(* PLC project Unnamed, Unknown Unnamed 1 *)
(* stored: creationDateTime 2025-10-16T09:35:51, modificationDateTime 2025-10-21T14:08:54 *)

PROGRAM motor_ctrl
  VAR
    motor_error AT %IX0.0 : BOOL;
    motor_error_true AT %IX0.1 : BOOL;
    run_motor AT %QX0.0 : BOOL;
    motor_running AT %QX0.1 : BOOL;
    stop_motor AT %QX0.2 : BOOL;
    run_motor_true AT %QX0.3 : BOOL;
    motor_running_true AT %QX0.4 : BOOL;
    stop_motor_true AT %QX0.5 : BOOL;
    motor_rpm AT %IW0 : INT;
    motor_rpm_true AT %IW1 : INT;
    target_freq AT %QW0 : INT;
    target_freq_true AT %QW1 : INT := 120;
  END_VAR
  VAR  (* added by the conversion: wires and edge detectors of the diagram *)
    R_TRIG1 : R_TRIG;
    R_TRIG2 : R_TRIG;
  END_VAR

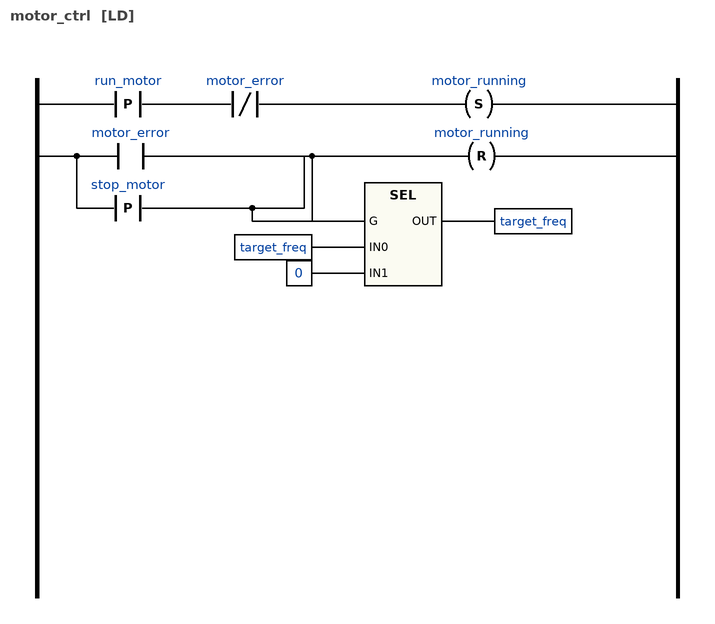
(* LD diagram, written out as Structured Text *)
R_TRIG1(CLK := run_motor);
IF R_TRIG1.Q AND NOT motor_error THEN motor_running := TRUE; END_IF;
R_TRIG2(CLK := stop_motor);
IF motor_error OR R_TRIG2.Q THEN motor_running := FALSE; END_IF;
target_freq := SEL(R_TRIG2.Q OR motor_error, target_freq, 0);
END_PROGRAM

CONFIGURATION Config0
  RESOURCE Res0 ON PLC
    TASK task0(INTERVAL := T#20ms, PRIORITY := 0);
    PROGRAM instance0 WITH task0 : motor_ctrl;
  END_RESOURCE
END_CONFIGURATION
